{attribute 'qualified_only'}
{attribute 'strict'}
TYPE PisaPulseCommMode :
(
	Offline :=0,
	Unidirectional := 1,
	Bidirectional :=2
	
);
END_TYPE

(* stored: Version 1.1.0.1, ProductVersion 3.1.4024.15
   EnumerationTextList PisaPulseCommMode: Id {0b59b537-bbea-4462-9656-d775a11b7295} *)
